FUNCTION_BLOCK Job IMPLEMENTS I_JobNode
VAR
	_iNext: I_JobNode;
	_iPrev: I_JobNode;
	_iWorker: I_Worker;
	_iTask: I_Job;
	_eState: TaskState;
END_VAR

PROPERTY INTERNAL _Next : I_JobNode
GET
_Next := _iNext;
END_GET
SET
_iNext := _Next;
END_SET
END_PROPERTY

PROPERTY INTERNAL _Prev : I_JobNode
GET
_Prev := _iPrev;
END_GET
SET
_iPrev := _Prev;
END_SET
END_PROPERTY

METHOD INTERNAL _Reset
_iNext := 0;
_iPrev := 0;
_eState := TaskState.Idle;
END_METHOD

METHOD INTERNAL _Run
VAR_INPUT
END_VAR
_eState := TaskState.Running;
_iTask.Run();
_eState := TaskState.Ready;
END_METHOD

METHOD Abort : Result
VAR_INPUT
END_VAR
IF _eState = TaskState.Idle THEN
	Abort := Err.IncArg;
	RETURN;
END_IF

_eState := TaskState.Aborted;
Abort := Ok;
END_METHOD

METHOD Complete : Result
VAR_INPUT
END_VAR
IF _eState <> TaskState.Running THEN
	Complete := Err.IncArg;
	RETURN;
END_IF

_eState := TaskState.Completed;
Complete := Ok;
END_METHOD

//FB_Init is always available implicitly and it is used primarily for initialization.
//The return value is not evaluated. For a specific influence, you can also declare the
//methods explicitly and provide additional code there with the standard initialization
//code. You can evaluate the return value.
METHOD FB_Init: BOOL
VAR_INPUT
    bInitRetains: BOOL; // TRUE: the retain variables are initialized (reset warm / reset cold)
    bInCopyCode: BOOL;  // TRUE: the instance will be copied to the copy code afterward (online change)
	iTask: I_Job;
END_VAR
_iTask := iTask;
IF _iTask = 0 THEN
	_eState := TaskState.Error;
END_IF
END_METHOD

METHOD Start : Result
VAR_INPUT
END_VAR
IF _eState <> TaskState.Idle THEN
	Start := Err.IncArg;
	RETURN;
END_IF

IF _iWorker = 0 THEN
	Start := Err.Itf0;
	RETURN;
END_IF

IF IsOk(_iWorker.Enqueue(THIS^), nOut => Start) THEN
	_eState := TaskState.Ready;
END_IF
END_METHOD

PROPERTY State : TaskState
GET
State := _eState;
END_GET
END_PROPERTY

PROPERTY Worker : I_Worker
GET
Worker := _iWorker;
END_GET
SET
IF _eState = TaskState.Idle THEN
	_iWorker := Worker;
END_IF
END_SET
END_PROPERTY

END_FUNCTION_BLOCK

(* stored: Version 1.1.0.1
   POU Job: Id {d189be26-c4d1-421c-b40d-0f9c5d388d23}, SpecialFunc None
   Folder _: Id {788cea3f-9c89-4c58-9f8b-26391a806f35}
   Folder Job: Id {30958162-07b8-4f88-92e6-ce23182d425b}
   Property _Next: Id {5e0a6afe-9bd8-403e-ae27-c1e3514413ad}
   Get Get: Id {56f40b47-08b4-4d87-acff-0407d2abd968}
   Set Set: Id {ce3e5deb-8114-42c1-92b7-0c5fd1201809}
   Property _Prev: Id {ab52e9e9-e1b8-4e36-a7cc-c3ffe7b8a011}
   Get Get: Id {e01b98b1-7d87-4f71-b8c9-d2aa7f7c1966}
   Set Set: Id {79a3a2b2-e6f3-4c9e-ab65-e3ea0bffc457}
   Method _Reset: Id {a0ed9277-faf0-472d-a5ff-d71c18d5c81a}
   Method _Run: Id {282b1123-78b3-4f76-80ac-354db08c0351}
   Method Abort: Id {c1b254d3-82b7-426a-bcdd-c337343702ca}
   Method Complete: Id {aabcf2a2-bc4a-433a-851b-c2329283fbd4}
   Method FB_Init: Id {6a9e7401-d8e2-47ed-9b55-404b5de36348}
   Method Start: Id {64d9d087-d2ba-4baf-8149-dc62e899d49b}
   Property State: Id {6447f694-df9c-483c-9624-6f2e9a8b97e7}
   Get Get: Id {bd91dcf6-8939-49c4-b291-29f8a1b3b103}
   Property Worker: Id {62c059a9-8170-459f-9379-8371a51c831c}
   Get Get: Id {927952be-4625-4ef1-867b-591ea7d3dec4}
   Set Set: Id {2b1cd96d-0301-44ad-89a4-fe218d4224f9} *)
